ABB RobotStudio station: BTL.rspag

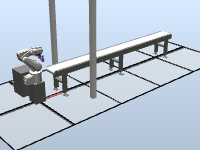
--- station ---
Station Solution14_1 (saved by RobotStudio 6.8.8307.1040)
Controller IRB_120_3kg_0.58m, task T_ROB1: task frame (RAPID world) sits at (4.2, 14.83, 360) mm in the station
Controller IRB_120_3kg_0.58m
  mechanical unit ROB_1: IRB120_3_58__01, 6 joints, base frame (0, 0, 0) mm
Layout (positions relative to the parent item):
  - IRB120_3_58__01 [mechanism, from Robots\IRB120_3_58_G_01.rslib] at (4.2, 14.83, 360) mm; joint values [0, -0.8727, 0.8727, 0, 1.5708, 0] (rad or m)
  - Suction_1 [mechanism] at (99.37, 14.83, 821.55) mm, rotated rx 180 ry 0 rz 180 deg
      TCP XP at (-62.25, 0.56, 103.67) mm
      links: suck
  - Part_2 [part] at (-95.8, -85.17, 0) mm
  - Convenyor Belt [smart component]
      signals: DO Do1
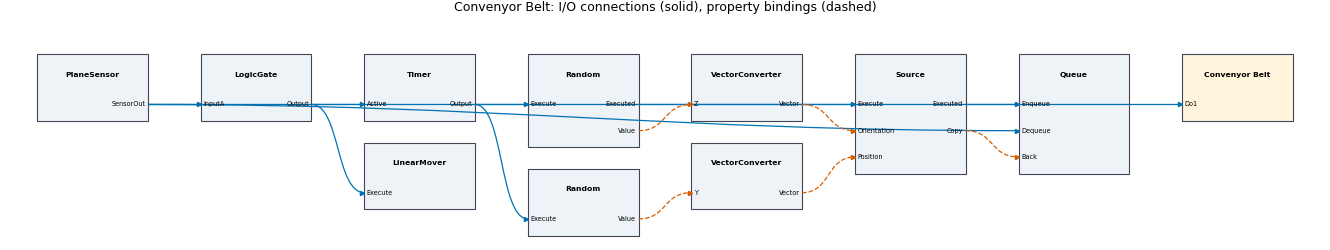
      connections:
        Timer.Output -> Random.Execute
        Random.Executed -> Source.Execute
        Source.Executed -> Queue.Enqueue
        PlaneSensor.SensorOut -> LogicGate.InputA
        PlaneSensor.SensorOut -> Queue.Dequeue
        LogicGate.Output -> LinearMover.Execute
        LogicGate.Output -> Timer.Active
        PlaneSensor.SensorOut -> Convenyor Belt.Do1
        Timer.Output -> Random.Execute
        Random.Value => VectorConverter.Z
        VectorConverter.Vector => Source.Orientation
        Source.Copy => Queue.Back
        VectorConverter.Vector => Source.Position
        Random.Value => VectorConverter.Y
    - Belt Conveyor [part] at (334.76, -134.1, 0) mm
    - matchbox [part] at (3268.53, 15, 15) mm
    - PlaneSensor [smart component, from Components\PlaneSensor.rslib]
        properties: Origin=[0.334765 0.165897 0.497]; Axis1=[0 0 0.05]; Axis2=[0 -0.3 0]; SensedPart=(none)
      - _sensorPart_ [part]
    - Timer [smart component, from Components\Timer.rslib]
        properties: StartTime=0; Interval=3.6; Repeat=true; CurrentTime=13.584
    - LinearMover [smart component, from Components\LinearMover.rslib]
        properties: Object=Queue; Direction=[-0.001 0 0]; Speed=0.2; Reference=Global; ReferenceObject=(none)
    - Source [smart component, from Components\Source.rslib]
        properties: Source=matchbox; Copy=(none); Parent=(none); Position=[3.268532 -0.0160380529919816 0.515388]; Orientation=[0 0 1.53910420828411]; Transient=false; PhysicsBehavior=0
    - Queue [smart component, from Components\Queue.rslib]
        properties: Back=(none); Front=(none); Queue={eaf5c064-27fd-41d6-82af-5ef21e71991e};{a3f5a395-1d45-4406-bcec-cae0d85dbb73};{613f6905-3ba6-4768-be48-6f95c265eb99};{0458d3b8-0919-4158-b7da-edfade52fce7};{166856ff-83ff-4faf-9608-c77b5b83d6b7};{74c26f46-fa4f-4ad3-ac73-7f6981861632};{c7b43b97-2bb4-4b75-9240-80eff27b8537};{a65cee13-cd64-4a50-81b2-256528f3d475};{6a8b7e73-c902-4c26-99f7-4df515df99b4};{212663d5-59b9-41ea-95fc-367cb3ff5d6f};{8f4e962d-8e0e-40f8-874f-b1b0542bcd40};{1eb5d92f-647c-4994-bada-8043b7148635};{e9dfa5d0-d6ef-464f-bf55-a1ba59cc24c6};{791a001c-0736-4f4a-9a75-d01a47d8fc11};{6378e3c8-a755-43c0-9d68-1e202f971c3a};{fcf3277e-53a4-4b94-9ad9-c831395550d6};{a380411a-908e-4b6f-afb5-b870898f272f}; NumberOfObjects=3
    - LogicGate [smart component, from Components\LogicGate.rslib]
        properties: Operator=NOT; Delay=0
    - VectorConverter [smart component, from Components\VectorConverter.rslib]
        properties: X=0; Y=0; Z=1.53910420828411; Vector=[0 0 1.53910420828411]
    - Random [smart component, from Components\Random.rslib]
        properties: Value=1.53910420828411; Min=-1.571; Max=1.571
    - VectorConverter [smart component, from Components\VectorConverter.rslib]
        properties: X=3.268532; Y=-0.0160380529919816; Z=0.515388; Vector=[3.268532 -0.0160380529919816 0.515388]
    - Random [smart component, from Components\Random.rslib]
        properties: Value=-0.0160380529919816; Min=-0.04; Max=0.06
  - Part_4 [part] at (-126.7, 276.91, 0) mm
  - RB_SUCK [smart component]
      signals: DI Di1
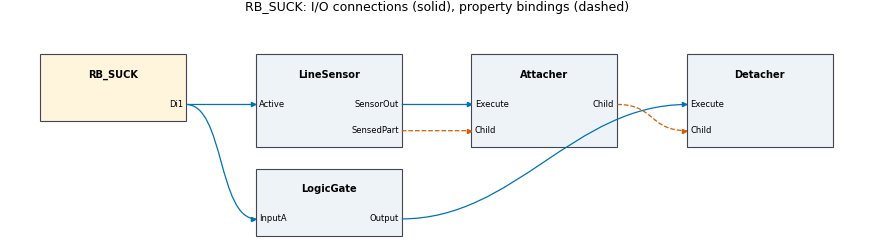
      connections:
        RB_SUCK.Di1 -> LineSensor.Active
        RB_SUCK.Di1 -> LogicGate.InputA
        LineSensor.SensorOut -> Attacher.Execute
        LogicGate.Output -> Detacher.Execute
        LineSensor.SensedPart => Attacher.Child
        Attacher.Child => Detacher.Child
    - Detacher [smart component, from Components\Detacher.rslib]
        properties: Child=(none); KeepPosition=true
    - Attacher [smart component, from Components\Attacher.rslib]
        properties: Parent=XP; Flange=0; Child=(none); Mount=true; Offset=[0 0 0]; Orientation=[0 0 0]
    - LineSensor [smart component, from Components\LineSensor.rslib] at (0, 0, 0) mm
        properties: Start=[0.161625 0.01539 0.722883]; End=[0.161625 0.01539 0.712883]; Radius=0.003; SensedPart=(none); SensedPoint=[0 0 0]
      - _sensorPart_ [part]
    - LogicGate [smart component, from Components\LogicGate.rslib]
        properties: Operator=NOT; Delay=0
  - CAMERA [smart component]
      signals: DI Di1
      connections:
        CAMERA.Di1 -> Camera.Execute
        CAMERA.Di1 -> LightControl.Enabled
    - Camera [graphiccomponentgroup] at (792.65, 47.53, 1993.8) mm, rotated rx 0 ry 0 rz -90 deg
      - Frame [part] at (0, 40, -1000) mm, rotated rx 90 ry 0 rz 0 deg
      - Camera [part] at (-1.73, 34.11, -243.83) mm, rotated rx 90 ry 0 rz 0 deg
    - LightControl [smart component, from Components\LightControl.rslib]
        properties: Light=Spotlight; Color=-128; CastShadows=true; AmbientIntensity=0; DiffuseIntensity=1; HighlightIntensity=0.900000035762787; SpotAngle=0.872664625997165; Range=0
    - Camera [smart component, from Components\Camera.rslib]
        properties: Path=C:\Users\Admin\Desktop\PY; File Name=pic
  - Frame_1 [frame]
  - Frame_3 [frame]
Attachment: Spotlight is attached to CAMERA
Attachment: Suction_1 is attached to IRB120_3_58__01 / Link6
Attachment: LineSensor is attached to IRB120_3_58__01 / Link6
Station logic (signal -> signal, property => property):
  Convenyor Belt.Do1 -> IRB_120_3kg_0.58m.Sensor
  IRB_120_3kg_0.58m.camera -> CAMERA.Di1
  IRB_120_3kg_0.58m.suck -> RB_SUCK.Di1
Targets, tools, work objects and paths stored in the station and not in the controller backup, written as RAPID:
! task T_ROB1
MODULE Module1
  CONST robtarget Target_40:=[[342.997624079,-23.608141871,147.887969085],[0.000000008,0,1,-0.000000001],[-1,-1,-1,0],[9E+09,9E+09,9E+09,9E+09,9E+09,9E+09]];
ENDMODULE


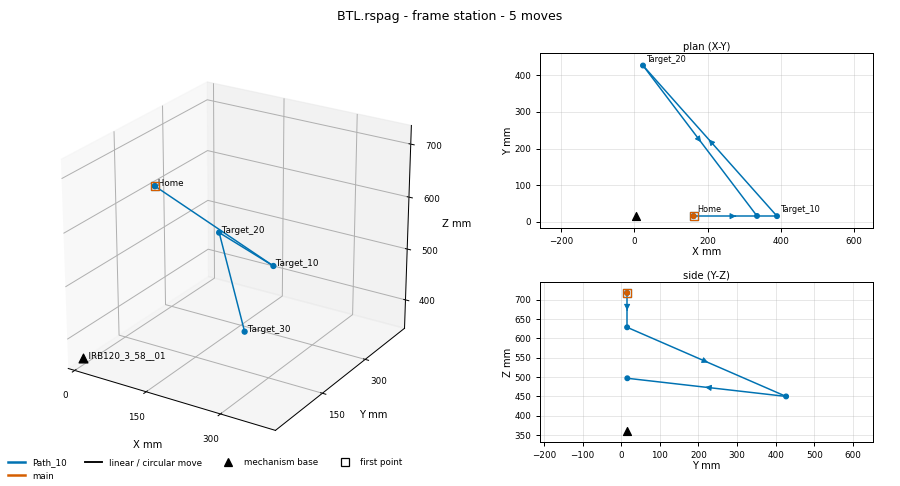
[picture p0: tool path of BTL.rspag in frame station, 5 of 11 moves have a stored position in this frame; points joined in program order, loops and branches not executed]
--- Backups/IRB_120_3kg_0.58m/RAPID/TASK1/PROGMOD/CalibData.mod ---
MODULE CalibData
	PERS tooldata XP:=[TRUE,[[-62.255,0.556,103.67],[1,0,0,0]],[1,[0,0,1],[1,0,0,0],0,0,0]];
ENDMODULE

--- Backups/IRB_120_3kg_0.58m/RAPID/TASK1/PROGMOD/Module1.mod ---
MODULE Module1
	CONST robtarget Home:=[[157.423000358,0.556,357.882654615],[0,0,1,0],[0,0,0,0],[9E+09,9E+09,9E+09,9E+09,9E+09,9E+09]];
	CONST robtarget Target_10:=[[385.179918373,0.556,268.935964011],[-0.000000104,0,1,0],[-1,-1,-1,0],[9E+09,9E+09,9E+09,9E+09,9E+09,9E+09]];
	CONST robtarget Target_20:=[[19.096656949,412.074903161,89.999961705],[-0.00000009,-0.000000042,1,0.000000014],[1,0,1,0],[9E+09,9E+09,9E+09,9E+09,9E+09,9E+09]];
    CONST robtarget Target_30:=[[330.56301599,1.062598023,136.999948682],[0.000000007,0,1,0.000000004],[0,0,0,0],[9E+09,9E+09,9E+09,9E+09,9E+09,9E+09]];
	PROC Path_10()
	    MoveL Home,v1000,z100,XP\WObj:=wobj0;
	    MoveL Target_10,v1000,z100,XP\WObj:=wobj0;
	    MoveL Target_20,v1000,z100,XP\WObj:=wobj0;
        MoveL Target_30,v1000,z100,XP\WObj:=wobj0;
	ENDPROC
ENDMODULE

--- Backups/IRB_120_3kg_0.58m/RAPID/TASK1/PROGMOD/VisionPick.mod ---
MODULE VisionPick

    ! ================== SOCKET ==================
    VAR socketdev srv;
    VAR socketdev cli;
    VAR string    msg;
    VAR string    val;

    VAR robtarget tPick;
    VAR robtarget tUp;

    VAR num count := 0;   ! d?m s? h?p dã x?p (0,1,2,...)
    VAR num col;
    VAR num row;
    VAR num layer;
    VAR num xOff;
    VAR num yOff;
    VAR num zOff;

    VAR robtarget origin;
    VAR robtarget tPlace;
    VAR robtarget tPlaceUp;

    ! K?t qu? vision (mm, deg)
    VAR num dx;
    VAR num dy;
    VAR num ang;

    ! Tham s? chung
    CONST string HOST := "127.0.0.1";
    CONST num    PORT := 11000;

    ! ================== HÀM LOG CMD SANG PYTHON ==================
    PROC LogCmd(string txt)
        ! G?i 1 dòng log: LOG:... + xu?ng dòng (ASCII 0x0A)
        SocketSend cli, \Str:="LOG:" + txt + "\0A";
    ENDPROC

    ! ================== MAIN ==================
    PROC main()
        ! T?o socket server trên ABB
        SocketCreate srv;
        SocketBind   srv, HOST, PORT;
        SocketListen srv;
        SocketAccept srv, cli;
        LogCmd("Python connected to vision socket");

        ! D?m b?o nh? hút ban d?u
        Reset suck;
        WaitTime 0.1;

        MoveJ Home, v1000, z50, XP\WObj:=wobj0;

        WHILE TRUE DO
            ! 1) D?i c?m bi?n báo có v?t
            WaitDI sensor, 1;
            LogCmd("Sensor ON - co vat");

            ! 2) B?t camera 0.5s (trigger ch?p ?nh)
            Set camera;
            WaitTime 0.5;
            Reset camera;
            LogCmd("Trigger camera xong");

            ! 3) G?i yêu c?u Python x? lý ?nh
            SocketSend cli, \Str:="CAPTURE" + "\0A";
            LogCmd("Gui CAPTURE cho Python");

            ! 4) Nh?n k?t qu? DX, DY, ANG t? Python
            ReceiveVisionResult;

            ! 5) G?i xác nh?n dã nh?n k?t qu?
            SocketSend cli, \Str:="OK_VISION" + "\0A";
            LogCmd("OK_VISION sent");

            ! 6) Th?c hi?n pick theo k?t qu? vision
            PickFromVision;

            ! 7) D?t v?t xu?ng v? trí x?p
            PlaceToTarget;

            ! 8) D?i sensor v? 0 tru?c vòng sau
            WaitDI sensor, 0;
            LogCmd("Sensor OFF - cho vong moi");
        ENDWHILE
    ENDPROC

    ! ================== NH?N K?T QU? T? PYTHON ==================
    PROC ReceiveVisionResult()
        VAR num gotDX;
        VAR num gotDY;
        VAR num gotANG;

        gotDX := 0;
        gotDY := 0;
        gotANG := 0;

        LogCmd("Cho ket qua vision...");

        WHILE (gotDX = 0) OR (gotDY = 0) OR (gotANG = 0) DO
            SocketReceive cli, \Str:=msg;
            LogCmd("RX:" + msg);

            ! DX:xxx
            IF (StrLen(msg) > 3) AND (StrPart(msg,1,3) = "DX:") THEN
                val := StrPart(msg, 4, StrLen(msg)-3);
                IF StrToVal(val, dx) THEN
                    LogCmd("DX=" + ValToStr(dx));
                    gotDX := 1;
                ELSE
                    LogCmd("ERR parse DX");
                ENDIF

            ! DY:yyy
            ELSEIF (StrLen(msg) > 3) AND (StrPart(msg,1,3) = "DY:") THEN
                val := StrPart(msg, 4, StrLen(msg)-3);
                IF StrToVal(val, dy) THEN
                    LogCmd("DY=" + ValToStr(dy));
                    gotDY := 1;
                ELSE
                    LogCmd("ERR parse DY");
                ENDIF

            ! ANG:zzz
            ELSEIF (StrLen(msg) > 4) AND (StrPart(msg,1,4) = "ANG:") THEN
                val := StrPart(msg, 5, StrLen(msg)-4);
                IF StrToVal(val, ang) THEN
                    LogCmd("ANG=" + ValToStr(ang));
                    gotANG := 1;
                ELSE
                    LogCmd("ERR parse ANG");
                ENDIF

            ELSE
                LogCmd("Message khac: " + msg);
            ENDIF
        ENDWHILE

        LogCmd("Da nhan day du DX, DY, ANG");
    ENDPROC

    ! ================== PICK T? K?T QU? VISION ==================
    PROC PickFromVision()
        VAR robtarget tBase;

        LogCmd("PickFromVision START");
        LogCmd("dx = " + ValToStr(dx));
        LogCmd("dy = " + ValToStr(dy));
        LogCmd("ang = " + ValToStr(ang));

        ! 1) Offset v? trí theo h? wobj (bang t?i):
        !    dx, dy là mm theo X, Y c?a wobj0
        tBase := Offs(Target_30, dx, -dy, 10.89);

        ! 2) Xoay TCP quanh tr?c Z (tool) n?u c?n
        tPick := RelTool(tBase, 0, 0, 0 \Rz:=ang);

        ! 3) Di?m trên cao
        tUp := Offs(tPick, 0, 0, 100);

        LogCmd("MoveJ len diem tren cao");
        MoveJ tUp, v1000, z50, XP\WObj:=wobj0;

        LogCmd("Ha xuong diem pick");
        MoveL tPick, v200, fine, XP\WObj:=wobj0;

        WaitTime 0.3;
        LogCmd("Bat suck");
        Set suck;
        WaitTime 0.3;

        LogCmd("Nhat len lai");
        MoveL tUp, v500, z50, XP\WObj:=wobj0;
    ENDPROC



    ! ================== PLACE T?I V? TRÍ X?P ==================
    PROC PlaceToTarget()
        origin := Offs(Target_20,-78,-48, 16);

        ! 3 c?t × 3 hàng trong 1 l?p, 9 h?p / l?p
        col   := count MOD 3;             ! 0..2
        row   := (count DIV 3) MOD 3;     ! 0..2
        layer := count DIV 9;             ! 0..?

        xOff := col   * 52;
        yOff := row   * 32;
        zOff := layer * 17;

        ! Tính di?m d?t và di?m trên cao
        tPlace   := Offs(origin,xOff,yOff, zOff);
        tPlaceUp := Offs(tPlace, 0, 0, 100);

        LogCmd("Den tren cao vi tri xep");
        MoveJ tPlaceUp, v1000, z50, XP\WObj:=wobj0;

        LogCmd("Ha xuong vi tri xep");
        MoveL tPlace, v200, fine, XP\WObj:=wobj0;

        LogCmd("Tat suck");
        Reset suck;
        WaitTime 0.3;

        LogCmd("Nhat len khoi vi tri xep");
        MoveL tPlaceUp, v500, z50, XP\WObj:=wobj0;

        ! Tang b? d?m - chuy?n sang ô ti?p theo
        count := count + 1;
        ! N?u mu?n reset khi d?y m?t pallet 3x3xN, ví d? 2 l?p:
        ! IF count >= 18 THEN
        !     count := 0;
        ! ENDIF
    ENDPROC


ENDMODULE

--- Backups/IRB_120_3kg_0.58m/SYSPAR/EIO.cfg ---
EIO:CFG_1.0:6:1::
#
EIO_SIGNAL:

      -Name "sensor" -SignalType "DI"

      -Name "camera" -SignalType "DO"

      -Name "suck" -SignalType "DO"
